// TwinCAT 3 PLC project VekSi_PLC
// ProgramVersion: 3.1.4026.22
// libraries:
//   Tc2_MC2, * (Beckhoff Automation GmbH)
//   Tc2_Standard, * (Beckhoff Automation GmbH)
//   Tc2_System, * (Beckhoff Automation GmbH)
//   Tc2_Utilities, * (Beckhoff Automation GmbH)
//   Tc3_IotBase, * (Beckhoff Automation GmbH)
//   Tc3_JsonXml, * (Beckhoff Automation GmbH)
// project tree:
//   Funtions/ FB_CSVLogger.TcPOU, FB_ValveControl.TcPOU (not stored), FB_MqttManager.TcPOU, MAIN.TcPOU
//   / PlcTask.TcTTO
//   State_Var/ E_CSVLogState.TcDUT, E_MqttManagerState.TcDUT, E_SystemState.TcDUT, E_ValveSource.TcDUT, E_ValveState.TcDUT, ST_MqttConfig.TcDUT, ST_MQTT_Command.TcDUT (not stored), ST_ValveData.TcDUT
//   Variables_Lists/ GVL_Config.TcGVL, GVL_HMI.TcGVL (not stored), GVL_IO.TcGVL, GVL_System.TcGVL (not stored)
// real-time tasks:
//   TASK PlcTask: cycle T#10ms, priority 20, ADS port 350
// motion (NC):
//   TASK NC-Task 1 SAF: cycle T#2ms, priority 4, ADS port 501
//   TASK NC-Task 1 SVB: cycle T#10ms, priority 8, ADS port 511
//   AXIS Axis 2 (id 2)
//     Dynamic: Acceleration=16.9085, Deceleration=16.9085, Jerk=53.5391
//     Velo: RefSearch=3, RefSync=3, SlowManual=3, FastManual=3, Fast=3, Maximum=6
//     OtherSettings: AllowMotionCmdToSlave=true
//     encoder EncType=1
//       EncPara: ScaleFactorNumerator=0.003048
//         Inc: RefSoftSyncMask=#x0000ffff, HomingSensorSource=1
//         TimeComp: TimeCompMode=1, EncDelayCycles=4
//     drive DrvType=24
//       Analog: VeloReferenz=6.096, TorqueSetpointScale=10, ScaleFactorActTorque=0.1
//       TimeComp: TaskDelayCycles=1
//     controller CtrType=1
//       CtrPara: PriorControlFactor=1
//         PosDiffControl: Enable=false
//         Observer: BandWidth=20
//   AXIS Axis 3 (id 3)
//     Dynamic: Acceleration=16.9085, Deceleration=16.9085, Jerk=53.5391
//     Velo: Maximum=6
//     OtherSettings: AllowMotionCmdToSlave=true
//     encoder EncType=1
//       EncPara: ScaleFactorNumerator=0.003048
//         Inc: RefSoftSyncMask=#x0000ffff
//         TimeComp: TimeCompMode=1, EncDelayCycles=4
//     drive DrvType=24
//       Analog: VeloReferenz=6.096, TorqueSetpointScale=10, ScaleFactorActTorque=0.1
//       TimeComp: TaskDelayCycles=1
//     controller CtrType=1
//       CtrPara: PriorControlFactor=1
//         PosDiffControl: Enable=false
//         Observer: BandWidth=20
//   AXIS Axis 1 (id 1)
//     Dynamic: Acceleration=16.9085, Deceleration=16.9085, Jerk=53.5391
//     Velo: RefSearch=3, RefSync=3, SlowManual=3, FastManual=3, Maximum=6
//     OtherSettings: AllowMotionCmdToSlave=true
//     encoder EncType=1
//       EncPara: ScaleFactorNumerator=0.003048
//         Inc: RefSearchInverse=true, RefSoftSyncMask=#x0000ffff
//         TimeComp: TimeCompMode=1, EncDelayCycles=4
//     drive DrvType=24
//       Analog: VeloReferenz=6.096, TorqueSetpointScale=10, ScaleFactorActTorque=0.1
//       TimeComp: TaskDelayCycles=1
//     controller CtrType=1
//       CtrPara: PriorControlFactor=1
//         PosDiffControl: Enable=false
//         Observer: BandWidth=20
// I/O:
//   DEVICE Device 1 (EtherCAT), AmsNetId 192.168.56.1.2.1
//     Term 1 (EK1200) [EK1200-5000 EtherCAT Power supply (2A E-Bus)]
//       Term 2 (EL6070-0033) [EL6070-0033 1Ch. Licence key terminal, individual licences]
//       Term 3 (EL1859) [EL1859 8Ch. Dig. Input 24V, 3ms, 8Ch. Dig. Output 24V, 0.5A]
//       Term 4 (EL3202) [EL3202 2Ch. Ana. Input PT100 (RTD)]
//       Term 5 (EL1004) [EL1004 4Ch. Dig. Input 24V, 3ms]
//       Term 6 (EL3074) [EL3074 4Ch. Ana. Input +/-10V, +/-20mA]
//       Term 7 (EK1322) [EK1322 2-port EtherCAT P junction with feed-in]
//         Box 8 (EPP7041-1002) [EPP7041-1002 1Ch. Stepper motor output stage (50V, 1.5A)]
//       Term 9 (EK1521-0010) [EK1521-0010 1 port EtherCAT junction (FX-SingleMode)]
//         Term 10 (EK1501-0010) [EK1501-0010 EtherCAT Coupler (2A E-Bus, FX-SingleMode, ID switch)]
//           Term 11 (EL3202) [EL3202 2Ch. Ana. Input PT100 (RTD)]
//           Term 12 (EL1859) [EL1859 8Ch. Dig. Input 24V, 3ms, 8Ch. Dig. Output 24V, 0.5A]
//           Term 13 (EL3074) [EL3074 4Ch. Ana. Input +/-10V, +/-20mA]
//           Term 22 (EL9011) [EL9011 End Terminal]
//       Term 14 (EK1521-0010) [EK1521-0010 1 port EtherCAT junction (FX-SingleMode)]
//         Term 15 (EK1501-0010) [EK1501-0010 EtherCAT Coupler (2A E-Bus, FX-SingleMode, ID switch)]
//           Term 16 (EL3202) [EL3202 2Ch. Ana. Input PT100 (RTD)]
//           Term 17 (EL1004) [EL1004 4Ch. Dig. Input 24V, 3ms]
//           Term 18 (EL3074) [EL3074 4Ch. Ana. Input +/-10V, +/-20mA]
//           Term 19 (EK1322) [EK1322 2-port EtherCAT P junction with feed-in]
//             Box 20 (EPP7041-1002) [EPP7041-1002 1Ch. Stepper motor output stage (50V, 1.5A)]
//             Box 21 (EPP7041-1002) [EPP7041-1002 1Ch. Stepper motor output stage (50V, 1.5A)]
// variable links:
//   NC-Task 1 SAF/Axes/Axis 1 <-> Device 1 (EtherCAT)/Term 1 (EK1200)/Term 7 (EK1322)/Box 8 (EPP7041-1002)
//     Drive/Inputs/In/nState1 @bit 3 <-> STM Status/Status/Error
//     Drive/Inputs/In/nState1 @bit 7 <-> STM Status/Status/Motor stall
//     Drive/Inputs/In/nState1 @bit 5 <-> STM Status/Status/Moving negative
//     Drive/Inputs/In/nState1 @bit 4 <-> STM Status/Status/Moving positive
//     Drive/Inputs/In/nState1 @bit 1 <-> STM Status/Status/Ready
//     Drive/Inputs/In/nState1 <-> STM Status/Status/Ready to enable
//     Drive/Inputs/In/nState1 @bit 6 <-> STM Status/Status/Torque reduced
//     Drive/Inputs/In/nState1 @bit 2 <-> STM Status/Status/Warning
//     Drive/Inputs/In/nState2 @bit 4 <-> STM Status/Status/Digital input 2
//     Drive/Inputs/In/nState2 @bit 5 <-> STM Status/Status/Sync error
//     Drive/Inputs/In/nState2 @bit 7 <-> STM Status/Status/TxPDO Toggle
//     Drive/Inputs/In/nState4 @bit 1 <-> WcState/InputToggle
//     Drive/Inputs/In/nState4 <-> WcState/WcState
//     Drive/Outputs/Out/nCtrl1 <-> STM Control/Control/Enable
//     Drive/Outputs/Out/nCtrl1 @bit 2 <-> STM Control/Control/Reduce torque
//     Drive/Outputs/Out/nCtrl1 @bit 1 <-> STM Control/Control/Reset
//     Drive/Outputs/Out/nCtrl2 @bit 3 <-> STM Control/Control/Digital output 1
//     Drive/Outputs/Out/nDataOut2[0] <-> STM Velocity/Velocity
//   NC-Task 1 SAF/Axes/Axis 2 <-> Device 1 (EtherCAT)/Term 1 (EK1200)/Term 14 (EK1521-0010)/Term 15 (EK1501-0010)/Term 19 (EK1322)/Box 20 (EPP7041-1002)
//     Drive/Inputs/In/nState1 @bit 3 <-> STM Status/Status/Error
//     Drive/Inputs/In/nState1 @bit 7 <-> STM Status/Status/Motor stall
//     Drive/Inputs/In/nState1 @bit 5 <-> STM Status/Status/Moving negative
//     Drive/Inputs/In/nState1 @bit 4 <-> STM Status/Status/Moving positive
//     Drive/Inputs/In/nState1 @bit 1 <-> STM Status/Status/Ready
//     Drive/Inputs/In/nState1 <-> STM Status/Status/Ready to enable
//     Drive/Inputs/In/nState1 @bit 6 <-> STM Status/Status/Torque reduced
//     Drive/Inputs/In/nState1 @bit 2 <-> STM Status/Status/Warning
//     Drive/Inputs/In/nState2 @bit 3 <-> STM Status/Status/Digital input 1
//     Drive/Inputs/In/nState2 @bit 4 <-> STM Status/Status/Digital input 2
//     Drive/Inputs/In/nState2 @bit 5 <-> STM Status/Status/Sync error
//     Drive/Inputs/In/nState2 @bit 7 <-> STM Status/Status/TxPDO Toggle
//     Drive/Inputs/In/nState4 @bit 1 <-> WcState/InputToggle
//     Drive/Inputs/In/nState4 <-> WcState/WcState
//     Drive/Outputs/Out/nCtrl1 <-> STM Control/Control/Enable
//     Drive/Outputs/Out/nCtrl1 @bit 2 <-> STM Control/Control/Reduce torque
//     Drive/Outputs/Out/nCtrl1 @bit 1 <-> STM Control/Control/Reset
//     Drive/Outputs/Out/nCtrl2 @bit 3 <-> STM Control/Control/Digital output 1
//     Drive/Outputs/Out/nDataOut2[0] <-> STM Velocity/Velocity
//     Enc/Inputs/In/nDataIn1[0] <-> ENC Status compact/Counter value
//     Enc/Inputs/In/nDataIn2[0] <-> ENC Status compact/Latch value
//     Enc/Inputs/In/nState1 @bit 4 <-> ENC Status compact/Status/Counter overflow
//     Enc/Inputs/In/nState1 @bit 3 <-> ENC Status compact/Status/Counter underflow
//     Enc/Inputs/In/nState1 @bit 7 <-> ENC Status compact/Status/Extrapolation stall
//     Enc/Inputs/In/nState1 <-> ENC Status compact/Status/Latch C valid
//     Enc/Inputs/In/nState1 @bit 1 <-> ENC Status compact/Status/Latch extern valid
//     Enc/Inputs/In/nState1 @bit 2 <-> ENC Status compact/Status/Set counter done
//     Enc/Inputs/In/nState2 @bit 4 <-> ENC Status compact/Status/Status of extern latch
//     Enc/Inputs/In/nState2 <-> ENC Status compact/Status/Status of input A
//     Enc/Inputs/In/nState2 @bit 1 <-> ENC Status compact/Status/Status of input B
//     Enc/Inputs/In/nState2 @bit 2 <-> ENC Status compact/Status/Status of input C
//     Enc/Inputs/In/nState2 @bit 5 <-> ENC Status compact/Status/Sync error
//     Enc/Inputs/In/nState2 @bit 7 <-> ENC Status compact/Status/TxPDO Toggle
//     Enc/Inputs/In/nState4 @bit 1 <-> WcState/InputToggle
//     Enc/Inputs/In/nState4 <-> WcState/WcState
//     Enc/Outputs/Out/nCtrl1 <-> ENC Control compact/Control/Enable latch C
//     Enc/Outputs/Out/nCtrl1 @bit 3 <-> ENC Control compact/Control/Enable latch extern on negative edge
//     Enc/Outputs/Out/nCtrl1 @bit 1 <-> ENC Control compact/Control/Enable latch extern on positive edge
//     Enc/Outputs/Out/nCtrl1 @bit 2 <-> ENC Control compact/Control/Set counter
//     Enc/Outputs/Out/nDataOut1[0] <-> ENC Control compact/Set counter value
//   NC-Task 1 SAF/Axes/Axis 3 <-> Device 1 (EtherCAT)/Term 1 (EK1200)/Term 14 (EK1521-0010)/Term 15 (EK1501-0010)/Term 19 (EK1322)/Box 21 (EPP7041-1002)
//     Drive/Inputs/In/nState1 @bit 3 <-> STM Status/Status/Error
//     Drive/Inputs/In/nState1 @bit 7 <-> STM Status/Status/Motor stall
//     Drive/Inputs/In/nState1 @bit 5 <-> STM Status/Status/Moving negative
//     Drive/Inputs/In/nState1 @bit 4 <-> STM Status/Status/Moving positive
//     Drive/Inputs/In/nState1 @bit 1 <-> STM Status/Status/Ready
//     Drive/Inputs/In/nState1 <-> STM Status/Status/Ready to enable
//     Drive/Inputs/In/nState1 @bit 6 <-> STM Status/Status/Torque reduced
//     Drive/Inputs/In/nState1 @bit 2 <-> STM Status/Status/Warning
//     Drive/Inputs/In/nState2 @bit 3 <-> STM Status/Status/Digital input 1
//     Drive/Inputs/In/nState2 @bit 4 <-> STM Status/Status/Digital input 2
//     Drive/Inputs/In/nState2 @bit 5 <-> STM Status/Status/Sync error
//     Drive/Inputs/In/nState2 @bit 7 <-> STM Status/Status/TxPDO Toggle
//     Drive/Inputs/In/nState4 @bit 1 <-> WcState/InputToggle
//     Drive/Inputs/In/nState4 <-> WcState/WcState
//     Drive/Outputs/Out/nCtrl1 <-> STM Control/Control/Enable
//     Drive/Outputs/Out/nCtrl1 @bit 2 <-> STM Control/Control/Reduce torque
//     Drive/Outputs/Out/nCtrl1 @bit 1 <-> STM Control/Control/Reset
//     Drive/Outputs/Out/nCtrl2 @bit 3 <-> STM Control/Control/Digital output 1
//     Drive/Outputs/Out/nDataOut2[0] <-> STM Velocity/Velocity
//     Enc/Inputs/In/nDataIn1[0] <-> ENC Status compact/Counter value
//     Enc/Inputs/In/nDataIn2[0] <-> ENC Status compact/Latch value
//     Enc/Inputs/In/nState1 @bit 4 <-> ENC Status compact/Status/Counter overflow
//     Enc/Inputs/In/nState1 @bit 3 <-> ENC Status compact/Status/Counter underflow
//     Enc/Inputs/In/nState1 @bit 7 <-> ENC Status compact/Status/Extrapolation stall
//     Enc/Inputs/In/nState1 <-> ENC Status compact/Status/Latch C valid
//     Enc/Inputs/In/nState1 @bit 1 <-> ENC Status compact/Status/Latch extern valid
//     Enc/Inputs/In/nState1 @bit 2 <-> ENC Status compact/Status/Set counter done
//     Enc/Inputs/In/nState2 @bit 4 <-> ENC Status compact/Status/Status of extern latch
//     Enc/Inputs/In/nState2 <-> ENC Status compact/Status/Status of input A
//     Enc/Inputs/In/nState2 @bit 1 <-> ENC Status compact/Status/Status of input B
//     Enc/Inputs/In/nState2 @bit 2 <-> ENC Status compact/Status/Status of input C
//     Enc/Inputs/In/nState2 @bit 5 <-> ENC Status compact/Status/Sync error
//     Enc/Inputs/In/nState2 @bit 7 <-> ENC Status compact/Status/TxPDO Toggle
//     Enc/Inputs/In/nState4 @bit 1 <-> WcState/InputToggle
//     Enc/Inputs/In/nState4 <-> WcState/WcState
//     Enc/Outputs/Out/nCtrl1 <-> ENC Control compact/Control/Enable latch C
//     Enc/Outputs/Out/nCtrl1 @bit 3 <-> ENC Control compact/Control/Enable latch extern on negative edge
//     Enc/Outputs/Out/nCtrl1 @bit 1 <-> ENC Control compact/Control/Enable latch extern on positive edge
//     Enc/Outputs/Out/nCtrl1 @bit 2 <-> ENC Control compact/Control/Set counter
//     Enc/Outputs/Out/nDataOut1[0] <-> ENC Control compact/Set counter value
//   VekSi_PLC/VekSi_PLC Instance <-> Device 1 (EtherCAT)/Term 1 (EK1200)/Term 7 (EK1322)/Box 8 (EPP7041-1002)
//     PlcTask Inputs/GVL_IO.bBottom_position_1 <-> STM Status/Status/Digital input 1
//   VekSi_PLC/VekSi_PLC Instance <-> NC-Task 1 SAF/Axes/Axis 1
//     PlcTask Inputs/MAIN.Axis_Valve1.NcToPlc <-> Outputs/ToPlc
//     PlcTask Outputs/MAIN.Axis_Valve1.PlcToNc <-> Inputs/FromPlc
//   VekSi_PLC/VekSi_PLC Instance <-> NC-Task 1 SAF/Axes/Axis 2
//     PlcTask Inputs/MAIN.Axis_Valve2.NcToPlc <-> Outputs/ToPlc
//     PlcTask Outputs/MAIN.Axis_Valve2.PlcToNc <-> Inputs/FromPlc
//   VekSi_PLC/VekSi_PLC Instance <-> NC-Task 1 SAF/Axes/Axis 3
//     PlcTask Inputs/MAIN.Axis_Valve3.NcToPlc <-> Outputs/ToPlc
//     PlcTask Outputs/MAIN.Axis_Valve3.PlcToNc <-> Inputs/FromPlc

CONFIGURATION VekSi_PLC
    RESOURCE PLC ON TwinCAT3
        TASK PlcTask(INTERVAL := T#10ms, PRIORITY := 20);
        PROGRAM MAIN WITH PlcTask : MAIN;
    END_RESOURCE
END_CONFIGURATION

// ---- State_Var/E_CSVLogState.TcDUT

// States:
//   CSV_IDLE        : Waiting for next log interval
//   CSV_PREPARE     : Build timestamp, filename, header/row strings
//   CSV_OPEN        : Open file in append mode
//   CSV_WRITE_HDR   : Write header (first row for new day in this PLC session)
//   CSV_WRITE_ROW   : Write one CSV data row
//   CSV_CLOSE       : Close file handle
//   CSV_ERROR       : Latch error until disabled or reset by logic
// ============================================================
TYPE E_CSVLogState :
(
    CSV_IDLE      := 0,
    CSV_PREPARE   := 1,
    CSV_OPEN      := 2,
    CSV_WRITE_HDR := 3,
    CSV_WRITE_ROW := 4,
    CSV_CLOSE     := 5,
    CSV_ERROR     := 6
);
END_TYPE

// ---- State_Var/E_MqttManagerState.TcDUT
{attribute 'strict'}
{attribute 'to_string'}
TYPE E_MqttManagerState :
(
    DISABLED        := 0,
    CONNECTING      := 1,
    CONNECTED       := 2,
    DISCONNECTING   := 3,
    WAIT_RECONNECT  := 4
);
END_TYPE

// ---- State_Var/E_SystemState.TcDUT
{attribute 'strict'}
{attribute 'to_string'}
TYPE E_SystemState :
(
    INIT             := 0,
    HOMING_REQUIRED  := 1,
    READY            := 2,
    RUN              := 3,
    FAULT            := 4
);
END_TYPE

// ---- State_Var/E_ValveSource.TcDUT
{attribute 'qualified_only'}
{attribute 'strict'}
{attribute 'to_string'}
TYPE E_ValveSource :
(
    NONE    := 0,   // No command received yet (startup default)
    HMI     := 1,   // Last setpoint was entered via local HMI
    MQTT    := 2    // Last setpoint was received via MQTT topic
);
END_TYPE

// ---- State_Var/E_ValveState.TcDUT
{attribute 'qualified_only'}
{attribute 'strict'}
{attribute 'to_string'}
TYPE E_ValveState :
(
    INIT    := 0,   // Initializing, powering axis
    HOMING  := 1,   // Performing homing sequence (MC_Home)
    IDLE    := 2,   // At position, no active command
    MOVING  := 3,   // MC_MoveAbsolute active, travelling to setpoint
	HALT	:= 4,
    HOLD    := 5,   // At setpoint, holding position
    FAULT   := 6,   // Error state — MC error, drive fault, or limit breach
    RESET   := 7    // Clearing fault, preparing to re-home
);
END_TYPE

// ---- State_Var/ST_MqttConfig.TcDUT
(*
  ST_MqttConfig
  =============
  Central MQTT runtime configuration structure.

  Project policy (this project):
  - Broker and topic settings are maintained in PLC code constants (GVL_Config).
  - HMI only enables/disables MQTT operation.
  - No broker parameter editing from HMI.
*)
TYPE ST_MqttConfig :
STRUCT
  (* ── Broker connection parameters ────────────────────────── *)
  sBrokerAddress  : STRING(255);   (* IP/hostname of broker                        *)
  nPort           : UINT;          (* 1883 = plain MQTT, 8883 = TLS (if enabled)   *)
  sClientId       : STRING(64);    (* Must be unique per broker                    *)
  sUsername       : STRING(64);    (* Optional                                      *)
  sPassword       : STRING(64);    (* Optional                                      *)
  bUseTls         : BOOL;          (* TRUE = secure transport (if broker supports)  *)

  (* ── Topic parameters ────────────────────────────────────── *)
  sTopicPrefix    : STRING(64);    (* Logical namespace, e.g. 'irrigation/site1'   *)
  sMainTopic      : STRING(128);   (* Status publish topic                          *)
  SubscribeTopic  : STRING(128);   (* Command subscribe topic                       *)

  (* ── Runtime timings ─────────────────────────────────────── *)
  tPublishInterval : TIME;         (* Periodic status publish interval              *)
  tReconnectDelay  : TIME;         (* Delay between reconnect attempts              *)
END_STRUCT
END_TYPE

// ---- State_Var/ST_ValveData.TcDUT

TYPE ST_ValveData :
STRUCT
    // --- Setpoints (written by HMI or MQTT) ---
    HMI_Setpoint    : REAL;         // Position setpoint from HMI (0.0–100.0 %)
    MQTT_Setpoint   : REAL;         // Position setpoint from MQTT (0.0–100.0 %)
    Active_Setpoint : REAL;         // Currently active setpoint (latest of HMI/MQTT)

    // --- Feedback (written by FB_ValveControl) ---
    Actual_Position : REAL;         // Actual valve position in % (from MC axis)
    Actual_Pos_Raw  : LREAL;        // Raw axis position in mm or steps (from MC2)

    // --- Command source tracking ---
    Source          : E_ValveSource;  // Who issued the last command
    MQTT_Enabled    : BOOL;           // Allow MQTT to override this valve's setpoint

    // --- State machine status ---
    State           : E_ValveState;  // Current state of FB_ValveControl
    IsHomed         : BOOL;          // TRUE once homing has been completed
    InPosition      : BOOL;          // TRUE when actual ≈ setpoint (within tolerance)
    IsFault         : BOOL;          // TRUE when in FAULT state
    FaultCode       : UDINT;         // MC or drive error code for diagnostics
	

	
    // --- Reset ---
    Reset_Cmd       : BOOL;          // HMI writes TRUE to request fault reset
END_STRUCT
END_TYPE

// ---- Variables_Lists/GVL_Config.TcGVL
{attribute 'qualified_only'}
VAR_GLOBAL CONSTANT
    // ── Valve motion parameters ───────────────────────────────
    VALVE_FULL_STROKE_MM           : REAL  := 6.096;     // Mechanical full travel for 0..100% scaling
    VALVE_POSITION_TOLERANCE       : REAL  := 0.5;       // In-position dead-band in percent
    VALVE_MOVE_VELOCITY            : LREAL := 1.5;       // mm/s
    VALVE_MOVE_ACCELERATION        : LREAL := 16.9085;   // mm/s²
    VALVE_MOVE_DECELERATION        : LREAL := 16.9085;   // mm/s²
    VALVE_MOVE_JERK                : LREAL := 53.5391;   // mm/s³
    VALVE_HOMING_VELOCITY          : LREAL := 1.0;       // Reference only (NC axis settings still apply)

    // ── CSV Logging ───────────────────────────────────────────
    CSV_LOG_INTERVAL_S             : TIME   := T#15M;
    CSV_FILE_PATH                  : STRING := 'C:\TwinCAT\3.1\Boot\Log\';
    CSV_FILENAME_PREFIX            : STRING := 'IrrigationLog_';

    // ── MQTT defaults (single source of truth) ───────────────
    // All MQTT configuration is centralized in this one constant structure.
    MQTT_CONFIG : ST_MqttConfig := (
        sBrokerAddress   := '192.168.1.100',
        nPort            := 1883,
        sClientId        := 'BeckhoffIrrigationPLC',
        sUsername        := '',
        sPassword        := '',
        bUseTls          := FALSE,
        sTopicPrefix     := 'irrigation',
        sMainTopic       := 'irrigation/status',
        SubscribeTopic   := 'irrigation/command',
        tPublishInterval := T#5M,
        tReconnectDelay  := T#30S
    );

    // ── Task cycle time ───────────────────────────────────────
    TASK_CYCLE_MS                  : UINT := 10;         // Must match TwinCAT task setting
END_VAR

// ---- Variables_Lists/GVL_IO.TcGVL
{attribute 'qualified_only'}
VAR_GLOBAL
	
	AI_L1V11  			: INT	:= -999 ;	// AT %I* // Water Level Sensors
	AI_L1V20  			: INT	:= -999 ;	// AT %I*
	AI_L2V21  			: INT	:= -999 ;	// AT %I*

	AI_Tmp_1 			: INT	:= -999;	// AT %I*
	AI_Tmp_2  			: INT	:= -999;	// AT %I*
	
	AI_PosFeedback_1	: INT	:= -999;	// AT %I* //Position feedback from the encoder
	AI_PosFeedback_2	: INT	:= -999;	// AT %I*
	AI_PosFeedback_3	: INT	:= -999;	// AT %I*
	

	bTop_position_1		AT %I*	: BOOL;
	bBottom_position_1	AT %I*	: BOOL;
END_VAR

// ---- Funtions/MAIN.TcPOU
PROGRAM MAIN
VAR
    // ── Valve function blocks (one instance per physical axis) ───────────────────
    fbValve1    : FB_ValveControl;
    fbValve2    : FB_ValveControl;
    fbValve3    : FB_ValveControl;

    // ── NC axis references ─────────────────────────────────────────────────────────
    // These variables must be linked to configured TwinCAT NC axes in I/O mapping.
    Axis_Valve1 : AXIS_REF;
    Axis_Valve2 : AXIS_REF;
    Axis_Valve3 : AXIS_REF;

    // ── Supporting modules ─────────────────────────────────────────────────────────
    fbCsvLogger   : FB_CsvLogger;
    fbMqttManager : FB_MqttManager;

    // ── MQTT runtime configuration ─────────────────────────────────────────────────
    // Initialized from GVL_Config once at startup. Fields may be changed in code
    // later if dynamic reconfiguration from HMI is added.
    stMqttConfig : ST_MqttConfig := (
        sBrokerAddress := GVL_Config.MQTT_DEFAULT_BROKER_IP,
        nPort := GVL_Config.MQTT_DEFAULT_PORT,
        sClientId := GVL_Config.MQTT_DEFAULT_CLIENT_ID,
        sUsername := GVL_Config.MQTT_DEFAULT_USERNAME,
        sPassword := GVL_Config.MQTT_DEFAULT_PASSWORD,
        sTopicPrefix := GVL_Config.MQTT_DEFAULT_TOPIC_PREFIX,
        sMainTopic := 'irrigation/status',
        SubscribeTopic := 'irrigation/command',
        tPublishInterval := T#5M,
        tReconnectDelay := T#30S
    );

    // ── Command arbitration helpers ────────────────────────────────────────────────
    // Stores previous HMI setpoints to detect operator changes.
    arrPrevHmiSetpoint : ARRAY[1..3] OF REAL := [-1.0, -1.0, -1.0];

    // Arrays passed directly to MQTT manager for compact status publishing.
    arrValveSetpoint : ARRAY[1..3] OF REAL;
    arrValveActual   : ARRAY[1..3] OF REAL;
    arrValveSource   : ARRAY[1..3] OF STRING(32);

    // Generic loop index used for repetitive valve operations.
    iValve : INT;
END_VAR

// =============================================================================
// SECTION 1 — READ HMI INPUTS AND CLAMP OPERATOR SETPOINTS
// =============================================================================
// LIMIT guarantees every valve command remains inside the configured legal range.
GVL_System.Valve[1].HMI_Setpoint := LIMIT(0.0, GVL_HMI.HMI_Valve1_Setpoint, 100.0);
GVL_System.Valve[2].HMI_Setpoint := LIMIT(0.0, GVL_HMI.HMI_Valve2_Setpoint, 100.0);
GVL_System.Valve[3].HMI_Setpoint := LIMIT(0.0, GVL_HMI.HMI_Valve3_Setpoint, 100.0);

GVL_System.Valve[1].Reset_Cmd := GVL_HMI.HMI_Valve1_Reset;
GVL_System.Valve[2].Reset_Cmd := GVL_HMI.HMI_Valve2_Reset;
GVL_System.Valve[3].Reset_Cmd := GVL_HMI.HMI_Valve3_Reset;

IF GVL_HMI.HMI_ResetAll THEN
    // Global reset request from HMI: pulse every valve reset command in this cycle.
    FOR iValve := 1 TO 3 DO
        GVL_System.Valve[iValve].Reset_Cmd := TRUE;
    END_FOR
    GVL_HMI.HMI_ResetAll := FALSE;
END_IF


// =============================================================================
// SECTION 2 — SETPOINT SOURCE ARBITRATION (HMI vs MQTT)
// =============================================================================
FOR iValve := 1 TO 3 DO
    // Startup fallback: if source is unknown, default to local HMI control.
    IF GVL_System.Valve[iValve].Source = E_ValveSource.NONE THEN
        GVL_System.Valve[iValve].Source := E_ValveSource.HMI;
        GVL_System.Valve[iValve].Active_Setpoint := GVL_System.Valve[iValve].HMI_Setpoint;
    END_IF

    // When operator changes HMI setpoint, HMI becomes authoritative source.
    IF ABS(GVL_System.Valve[iValve].HMI_Setpoint - arrPrevHmiSetpoint[iValve]) > 0.001 THEN
        GVL_System.Valve[iValve].Active_Setpoint := GVL_System.Valve[iValve].HMI_Setpoint;
        GVL_System.Valve[iValve].Source := E_ValveSource.HMI;
        arrPrevHmiSetpoint[iValve] := GVL_System.Valve[iValve].HMI_Setpoint;
    END_IF

    // Build compact telemetry arrays once here (reused by MQTT manager call).
    arrValveSetpoint[iValve] := GVL_System.Valve[iValve].Active_Setpoint;
    arrValveActual[iValve] := GVL_System.Valve[iValve].Actual_Position;
    arrValveSource[iValve] := TO_STRING(GVL_System.Valve[iValve].Source);
END_FOR


// =============================================================================
// SECTION 3 — MQTT CLIENT HANDLING
// =============================================================================
fbMqttManager (
    bEnable               := GVL_HMI.HMI_MQTT_bEnable,
    stConfig              := stMqttConfig,
    bApplyConfig          := FALSE,
    bPublish              := GVL_HMI.HMI_MQTT_mPublish,
    sPubTopic             := stMqttConfig.sMainTopic,
    sPubPayload           := '',
    bSubscribe            := GVL_HMI.HMI_MQTT_bEnable,
    sSubTopic             := stMqttConfig.SubscribeTopic,
    bUnsubscribe          := FALSE,
    sUnsubTopic           := '',
    bEnableStatusPublish  := GVL_HMI.HMI_MQTT_bEnable,
    tStatusPublishTime    := T#5M,
    sStatusTopic          := stMqttConfig.sMainTopic,
    rValveSetpoint        := arrValveSetpoint,
    rValveActual          := arrValveActual,
    sValveSource          := arrValveSource,
    rTemperature_C        := INT_TO_REAL(GVL_IO.AI_Tmp_1),
    rWaterLevel_Percent   := INT_TO_REAL(GVL_IO.AI_L1V11),
    sTimestamp            := DT_TO_STRING(CURRENT_DT())
);

IF fbMqttManager.bNewRemoteCommand AND GVL_HMI.HMI_MQTT_bEnable THEN
    // Remote command became valid in this cycle. Clamp values for safety before use.
    FOR iValve := 1 TO 3 DO
        GVL_System.Valve[iValve].MQTT_Setpoint := LIMIT(0.0, fbMqttManager.rMqttValveSetpoint[iValve], 100.0);
        GVL_System.Valve[iValve].Active_Setpoint := GVL_System.Valve[iValve].MQTT_Setpoint;
        GVL_System.Valve[iValve].Source := E_ValveSource.MQTT;
    END_FOR
END_IF


// =============================================================================
// SECTION 4 — EXECUTE PER-VALVE CONTROL FBs
// =============================================================================
// NOTE: Each valve FB is explicit to keep wiring to dedicated HMI tags readable.

// ── Valve 1 ────────────────────────────────────────────────────────────────────
fbValve1(
    Axis            := Axis_Valve1,
    HMI_Setpoint    := GVL_System.Valve[1].HMI_Setpoint,
    MQTT_Setpoint   := GVL_System.Valve[1].MQTT_Setpoint,
    MQTT_Enabled    := GVL_HMI.HMI_MQTT_bEnable,
    Enable          := TRUE,
    eHomingSelection := MC_Direct,
    Reset           := GVL_System.Valve[1].Reset_Cmd,
    MoveVelocity    := GVL_Config.VALVE_MOVE_VELOCITY,
    MoveAccel       := GVL_Config.VALVE_MOVE_ACCELERATION,
    MoveDecel       := GVL_Config.VALVE_MOVE_DECELERATION,
    MoveJerk        := GVL_Config.VALVE_MOVE_JERK,
    HomeVelocity    := GVL_Config.VALVE_HOMING_VELOCITY,
    FullStroke_mm   := GVL_Config.VALVE_FULL_STROKE_MM,
    PosTolerance    := GVL_Config.VALVE_POSITION_TOLERANCE,
    Move_Stop       := GVL_HMI.HMI_Valve1_Stop,
    UPDATE          := GVL_HMI.HMI_UPDATE,
    ZeroPosition    := GVL_IO.bBottom_position_1,
    bHoming         := GVL_HMI.HMI_Valve1_Homing,

    Actual_Position => GVL_System.Valve[1].Actual_Position,
    State           => GVL_System.Valve[1].State,
    Source          => GVL_System.Valve[1].Source,
    IsHomed         => GVL_System.Valve[1].IsHomed,
    InPosition      => GVL_System.Valve[1].InPosition,
    IsFault         => GVL_System.Valve[1].IsFault,
    FaultCode       => GVL_System.Valve[1].FaultCode,

    rTarget_mm      => GVL_HMI.Raw_Valve1_Setpoint,
    rActual_mm      => GVL_HMI.Raw_Valve1_Position
);

// ── Valve 2 ────────────────────────────────────────────────────────────────────
fbValve2(
    Axis            := Axis_Valve2,
    HMI_Setpoint    := GVL_System.Valve[2].HMI_Setpoint,
    MQTT_Setpoint   := GVL_System.Valve[2].MQTT_Setpoint,
    MQTT_Enabled    := GVL_HMI.HMI_MQTT_bEnable,
    Enable          := TRUE,
    eHomingSelection := MC_Direct,
    Reset           := GVL_System.Valve[2].Reset_Cmd,
    MoveVelocity    := GVL_Config.VALVE_MOVE_VELOCITY,
    MoveAccel       := GVL_Config.VALVE_MOVE_ACCELERATION,
    MoveDecel       := GVL_Config.VALVE_MOVE_DECELERATION,
    MoveJerk        := GVL_Config.VALVE_MOVE_JERK,
    HomeVelocity    := GVL_Config.VALVE_HOMING_VELOCITY,
    FullStroke_mm   := GVL_Config.VALVE_FULL_STROKE_MM,
    PosTolerance    := GVL_Config.VALVE_POSITION_TOLERANCE,
    Move_Stop       := GVL_HMI.HMI_Valve2_Stop,
    UPDATE          := GVL_HMI.HMI_UPDATE,
    bHoming         := GVL_HMI.HMI_Valve2_Homing,

    Actual_Position => GVL_System.Valve[2].Actual_Position,
    State           => GVL_System.Valve[2].State,
    Source          => GVL_System.Valve[2].Source,
    IsHomed         => GVL_System.Valve[2].IsHomed,
    InPosition      => GVL_System.Valve[2].InPosition,
    IsFault         => GVL_System.Valve[2].IsFault,
    FaultCode       => GVL_System.Valve[2].FaultCode,

    rTarget_mm      => GVL_HMI.Raw_Valve2_Setpoint,
    rActual_mm      => GVL_HMI.Raw_Valve2_Position
);

// ── Valve 3 ────────────────────────────────────────────────────────────────────
fbValve3(
    Axis            := Axis_Valve3,
    HMI_Setpoint    := GVL_System.Valve[3].HMI_Setpoint,
    MQTT_Setpoint   := GVL_System.Valve[3].MQTT_Setpoint,
    MQTT_Enabled    := GVL_HMI.HMI_MQTT_bEnable,
    Enable          := TRUE,
    eHomingSelection := MC_Direct,
    Reset           := GVL_System.Valve[3].Reset_Cmd,
    MoveVelocity    := GVL_Config.VALVE_MOVE_VELOCITY,
    MoveAccel       := GVL_Config.VALVE_MOVE_ACCELERATION,
    MoveDecel       := GVL_Config.VALVE_MOVE_DECELERATION,
    MoveJerk        := GVL_Config.VALVE_MOVE_JERK,
    HomeVelocity    := GVL_Config.VALVE_HOMING_VELOCITY,
    FullStroke_mm   := GVL_Config.VALVE_FULL_STROKE_MM,
    PosTolerance    := GVL_Config.VALVE_POSITION_TOLERANCE,
    Move_Stop       := GVL_HMI.HMI_Valve3_Stop,
    UPDATE          := GVL_HMI.HMI_UPDATE,
    bHoming         := GVL_HMI.HMI_Valve3_Homing,

    Actual_Position => GVL_System.Valve[3].Actual_Position,
    State           => GVL_System.Valve[3].State,
    Source          => GVL_System.Valve[3].Source,
    IsHomed         => GVL_System.Valve[3].IsHomed,
    InPosition      => GVL_System.Valve[3].InPosition,
    IsFault         => GVL_System.Valve[3].IsFault,
    FaultCode       => GVL_System.Valve[3].FaultCode,

    rTarget_mm      => GVL_HMI.Raw_Valve3_Setpoint,
    rActual_mm      => GVL_HMI.Raw_Valve3_Position
);


// =============================================================================
// SECTION 5 — CSV LOGGER EXECUTION
// =============================================================================
fbCsvLogger(
    bEnable              := TRUE,
    bForceWrite          := GVL_HMI.WriteTrigger,
    tLogInterval         := GVL_Config.CSV_LOG_INTERVAL_S,
    sBasePath            := GVL_Config.CSV_FILE_PATH,
    sPrefix              := GVL_Config.CSV_FILENAME_PREFIX,
    stValve              := GVL_System.Valve,
    rWaterLevel_Percent  := INT_TO_REAL(GVL_IO.AI_L1V11),
    rTemperature_C       := INT_TO_REAL(GVL_IO.AI_Tmp_1),

    dtLastWrite          => GVL_System.CSV_LastWriteTime,
    bError               => GVL_System.CSV_FileError,
    sCurrentFilename     => GVL_System.CSV_CurrentFile,
    eState               => GVL_System.CSV_LoggerState
);


// =============================================================================
// SECTION 6 — CLEANUP + HMI MIRRORING
// =============================================================================
// Reset commands are pulse-based: clear them after handing to FBs.
FOR iValve := 1 TO 3 DO
    GVL_System.Valve[iValve].Reset_Cmd := FALSE;
END_FOR
GVL_HMI.HMI_Valve1_Reset := FALSE;
GVL_HMI.HMI_Valve2_Reset := FALSE;
GVL_HMI.HMI_Valve3_Reset := FALSE;

// Copy valve runtime status to HMI tags.
GVL_HMI.ACT_Valve1_Position  := GVL_System.Valve[1].Actual_Position;
GVL_HMI.ACT_Valve1_State     := GVL_System.Valve[1].State;
GVL_HMI.ACT_Valve1_Source    := GVL_System.Valve[1].Source;
GVL_HMI.ACT_Valve1_Fault     := GVL_System.Valve[1].IsFault;
GVL_HMI.ACT_Valve1_FaultCode := GVL_System.Valve[1].FaultCode;

GVL_HMI.ACT_Valve2_Position  := GVL_System.Valve[2].Actual_Position;
GVL_HMI.ACT_Valve2_State     := GVL_System.Valve[2].State;
GVL_HMI.ACT_Valve2_Source    := GVL_System.Valve[2].Source;
GVL_HMI.ACT_Valve2_Fault     := GVL_System.Valve[2].IsFault;
GVL_HMI.ACT_Valve2_FaultCode := GVL_System.Valve[2].FaultCode;

GVL_HMI.ACT_Valve3_Position  := GVL_System.Valve[3].Actual_Position;
GVL_HMI.ACT_Valve3_State     := GVL_System.Valve[3].State;
GVL_HMI.ACT_Valve3_Source    := GVL_System.Valve[3].Source;
GVL_HMI.ACT_Valve3_Fault     := GVL_System.Valve[3].IsFault;
GVL_HMI.ACT_Valve3_FaultCode := GVL_System.Valve[3].FaultCode;

// System readiness is true only when all valves are homed and fault free.
GVL_System.AnyFaultActive :=
    GVL_System.Valve[1].IsFault OR
    GVL_System.Valve[2].IsFault OR
    GVL_System.Valve[3].IsFault;

GVL_System.SystemReady :=
    GVL_System.Valve[1].IsHomed AND
    GVL_System.Valve[2].IsHomed AND
    GVL_System.Valve[3].IsHomed AND
    NOT GVL_System.AnyFaultActive;

GVL_HMI.ACT_SystemReady := GVL_System.SystemReady;

END_PROGRAM

// ---- Funtions/FB_CSVLogger.TcPOU
(*  FB_CsvLogger
  ============
  Writes valve and sensor snapshots to CSV files on the IPC filesystem.

  File naming:
    <BasePath><Prefix><YYYY-MM-DD>.csv
  Example:
    C:\TwinCAT\IrrigationLogs\Irrigation_2026-04-28.csv

  Why a state machine?
    TwinCAT file function blocks are asynchronous (non-blocking). Each file
    action may require several PLC cycles to complete. This FB advances through
    explicit states so it remains deterministic and easy to troubleshoot.
*)

FUNCTION_BLOCK FB_CsvLogger

VAR_INPUT
  bEnable              : BOOL := TRUE;
  bForceWrite          : BOOL;          (* Rising edge = write one row immediately    *)
  tLogInterval         : TIME;          (* Periodic write interval                     *)
  sBasePath            : STRING(128);   (* Folder path including trailing '\'         *)
  sPrefix              : T_MaxString;   (* File prefix, e.g. 'Irrigation_'             *)
  stValve              : ARRAY[1..3] OF ST_ValveData;
  rWaterLevel_Percent  : REAL;
  rTemperature_C       : REAL;
END_VAR

VAR_OUTPUT
  bBusy                : BOOL;
  bError               : BOOL;
  nErrorCode           : UDINT;
  bFileExists          : BOOL := FALSE;
  dtLastWrite          : DT;
  sCurrentFile         : STRING(128);
  sCurrentFilename     : STRING(128);
  eState               : E_CSVLogState := E_CSVLogState.CSV_IDLE;
END_VAR

VAR
  (* ── File I/O FBs ───────────────────────────────────────── *)
  fbFileOpen           : FB_FileOpen;
  fbFileWrite          : FB_FileWrite;
  fbFileClose          : FB_FileClose;
  fbEnum               : FB_EnumFindFileEntry;

  hFilenumber          : UINT;
  cbLen                : UDINT;

  (* ── Trigger handling ───────────────────────────────────── *)
  tIntervalTimer       : TON;
  rtForceWrite         : R_TRIG;
  bTriggerWrite        : BOOL;

  (* ── Time/date helpers ──────────────────────────────────── *)
  fbGetTime            : FB_LocalSystemTime;
  nYear                : UINT;
  nMonth               : UINT;
  nDay                 : UINT;
  sYear                : STRING(8);
  sMonth               : STRING(4);
  sDay                 : STRING(4);

  (* ── CSV string buffers ─────────────────────────────────── *)
  sLine                : STRING(512);
  sHeader              : STRING(512);
  sSource              : STRING(8);

  (* ── Internal state helpers ─────────────────────────────── *)
  bEnumStart           : BOOL;
END_VAR

(* ============================================================
   SECTION 1 — CYCLIC HOUSEKEEPING
   ============================================================ *)
fbGetTime(bEnable := TRUE, dwCycle := 1);

// If logger is disabled, remain safe and idle.
IF NOT bEnable THEN
  tIntervalTimer(IN := FALSE);
  bTriggerWrite := FALSE;
  bBusy := FALSE;

  IF hFilenumber <> 0 THEN
    // Close any leftover open file handle before returning to idle.
    fbFileClose(hFile := hFilenumber, bExecute := TRUE);
    IF NOT fbFileClose.bBusy THEN
      fbFileClose(bExecute := FALSE);
      hFilenumber := 0;
    END_IF
  END_IF

  eState := E_CSVLogState.CSV_IDLE;
  RETURN;
END_IF

rtForceWrite(CLK := bForceWrite);
tIntervalTimer(IN := TRUE, PT := tLogInterval);

bTriggerWrite := rtForceWrite.Q OR tIntervalTimer.Q;

IF tIntervalTimer.Q THEN
  // Retrigger periodic timer after each elapsed interval.
  tIntervalTimer(IN := FALSE);
END_IF


(* ============================================================
   SECTION 2 — LOGGER STATE MACHINE
   ============================================================ *)
CASE eState OF

  E_CSVLogState.CSV_IDLE:
    bBusy := FALSE;

    IF bTriggerWrite THEN
      bError := FALSE;
      nErrorCode := 0;
      bFileExists := FALSE;
      bEnumStart := TRUE;
      eState := E_CSVLogState.CSV_PREPARE;
    END_IF


  E_CSVLogState.CSV_PREPARE:
    // Build filename as Prefix + YYYY-MM-DD.csv (daily file rotation).
    nYear  := fbGetTime.systemTime.wYear;
    nMonth := fbGetTime.systemTime.wMonth;
    nDay   := fbGetTime.systemTime.wDay;

    sYear  := UINT_TO_STRING(nYear);
    sMonth := UINT_TO_STRING(nMonth);
    sDay   := UINT_TO_STRING(nDay);

    IF nMonth < 10 THEN
      sMonth := CONCAT('0', sMonth);
    END_IF

    IF nDay < 10 THEN
      sDay := CONCAT('0', sDay);
    END_IF

    sCurrentFilename := sPrefix;
    sCurrentFilename := CONCAT(sCurrentFilename, sYear);
    sCurrentFilename := CONCAT(sCurrentFilename, '-');
    sCurrentFilename := CONCAT(sCurrentFilename, sMonth);
    sCurrentFilename := CONCAT(sCurrentFilename, '-');
    sCurrentFilename := CONCAT(sCurrentFilename, sDay);
    sCurrentFilename := CONCAT(sCurrentFilename, '.csv');

    sCurrentFile := CONCAT(sBasePath, sCurrentFilename);

    // Determine whether file already exists (header needed only for new files).
    IF bEnumStart THEN
      fbEnum(
        sPathName := sCurrentFile,
        eCmd := eEnumCmd_First,
        bExecute := TRUE,
        tTimeout := T#2S
      );
      bEnumStart := FALSE;
    ELSE
      fbEnum(bExecute := FALSE);
    END_IF

    IF NOT fbEnum.bBusy THEN
      fbEnum(bExecute := FALSE);

      IF (NOT fbEnum.bError) AND (fbEnum.stFindFile.sFileName <> '') THEN
        bFileExists := TRUE;
      ELSE
        bFileExists := FALSE;
      END_IF

      eState := E_CSVLogState.CSV_OPEN;
    END_IF


  E_CSVLogState.CSV_OPEN:
    bBusy := TRUE;

    fbFileOpen(
      sPathName := sCurrentFile,
      nMode     := FOPEN_MODEAPPEND,
      bExecute  := TRUE,
      hFile     => hFilenumber
    );

    IF NOT fbFileOpen.bBusy THEN
      fbFileOpen(bExecute := FALSE);

      IF fbFileOpen.bError THEN
        nErrorCode := fbFileOpen.nErrId;
        bError := TRUE;
        eState := E_CSVLogState.CSV_ERROR;
      ELSE
        hFilenumber := fbFileOpen.hFile;

        IF bFileExists THEN
          eState := E_CSVLogState.CSV_WRITE_ROW;
        ELSE
          eState := E_CSVLogState.CSV_WRITE_HDR;
        END_IF
      END_IF
    END_IF


  E_CSVLogState.CSV_WRITE_HDR:
    // Header is written exactly once per newly created daily file.
    sHeader := 'Timestamp,V1_Setpoint_%,V1_Actual_%,V1_Source,V2_Setpoint_%,V2_Actual_%,V2_Source,V3_Setpoint_%,V3_Actual_%,V3_Source,WaterLevel_%,Temperature_C$R$N';
    cbLen := INT_TO_UDINT(LEN(sHeader));

    fbFileWrite(
      bExecute   := TRUE,
      hFile      := hFilenumber,
      pWriteBuff := ADR(sHeader),
      cbWriteLen := cbLen
    );

    IF NOT fbFileWrite.bBusy THEN
      fbFileWrite(bExecute := FALSE);

      IF fbFileWrite.bError THEN
        nErrorCode := fbFileWrite.nErrId;
        bError := TRUE;
        eState := E_CSVLogState.CSV_CLOSE;
      ELSE
        eState := E_CSVLogState.CSV_WRITE_ROW;
      END_IF
    END_IF


  E_CSVLogState.CSV_WRITE_ROW:
    // Compose one CSV line from the latest process snapshot.
    sLine := CONCAT(SYSTEMTIME_TO_STRING(fbGetTime.systemTime), ',');

    sLine := CONCAT(sLine, CONCAT(REAL_TO_STRING(stValve[1].Active_Setpoint), ','));
    sLine := CONCAT(sLine, CONCAT(REAL_TO_STRING(stValve[1].Actual_Position), ','));
    sSource := TO_STRING(stValve[1].Source);
    sLine := CONCAT(sLine, CONCAT(sSource, ','));

    sLine := CONCAT(sLine, CONCAT(REAL_TO_STRING(stValve[2].Active_Setpoint), ','));
    sLine := CONCAT(sLine, CONCAT(REAL_TO_STRING(stValve[2].Actual_Position), ','));
    sSource := TO_STRING(stValve[2].Source);
    sLine := CONCAT(sLine, CONCAT(sSource, ','));

    sLine := CONCAT(sLine, CONCAT(REAL_TO_STRING(stValve[3].Active_Setpoint), ','));
    sLine := CONCAT(sLine, CONCAT(REAL_TO_STRING(stValve[3].Actual_Position), ','));
    sSource := TO_STRING(stValve[3].Source);
    sLine := CONCAT(sLine, CONCAT(sSource, ','));

    sLine := CONCAT(sLine, CONCAT(REAL_TO_STRING(rWaterLevel_Percent), ','));
    sLine := CONCAT(sLine, CONCAT(REAL_TO_STRING(rTemperature_C), '$R$N'));

    cbLen := INT_TO_UDINT(LEN(sLine));

    fbFileWrite(
      bExecute   := TRUE,
      hFile      := hFilenumber,
      pWriteBuff := ADR(sLine),
      cbWriteLen := cbLen
    );

    IF NOT fbFileWrite.bBusy THEN
      fbFileWrite(bExecute := FALSE);

      IF fbFileWrite.bError THEN
        nErrorCode := fbFileWrite.nErrId;
        bError := TRUE;
      ELSE
        bError := FALSE;
        dtLastWrite := SYSTEMTIME_TO_DT(fbGetTime.systemTime);
      END_IF

      eState := E_CSVLogState.CSV_CLOSE;
    END_IF


  E_CSVLogState.CSV_CLOSE:
    fbFileClose(hFile := hFilenumber, bExecute := TRUE);

    IF NOT fbFileClose.bBusy THEN
      fbFileClose(bExecute := FALSE);
      hFilenumber := 0;
      bBusy := FALSE;
      eState := E_CSVLogState.CSV_IDLE;
    END_IF


  E_CSVLogState.CSV_ERROR:
    bBusy := FALSE;
    bError := TRUE;

    // Recovery strategy: on next trigger, retry from preparation phase.
    IF bTriggerWrite THEN
      eState := E_CSVLogState.CSV_PREPARE;
    END_IF

END_CASE

END_FUNCTION_BLOCK

// ---- Funtions/FB_MqttManager.TcPOU
(*
============================================================
FUNCTION_BLOCK: FB_MqttManager
============================================================

PURPOSE
  Central MQTT manager for irrigation system.

  NOVICE SUMMARY
  - Think of this FB as a communication gateway between PLC and broker.
  - It handles connect/reconnect and topic subscription lifecycle.
  - It converts incoming JSON command payload into valve setpoints.
  - It builds outgoing JSON status payload from PLC runtime values.

HANDLES
  • MQTT connection / reconnection
  • Topic subscription / unsubscription
  • Manual publish
  • Cyclic JSON status publish
  • Incoming JSON command parsing
  • List of currently subscribed topics for HMI

EXPECTED INCOMING JSON
  {
    "valve_1": 25.0,
    "valve_2": 50.0,
    "valve_3": 75.0
  }

OUTGOING JSON
  Similar to CSV row:
    timestamp,
    valve setpoints,
    valve actual positions,
    valve command sources,
    temperature,
    water level

LIBRARIES
  • TF6701 / Tc3_IotBase
  • Tc2_Standard
============================================================
*)

FUNCTION_BLOCK FB_MqttManager
VAR_INPUT
    (* ── Connection control ───────────────────────────── *)
    bEnable         : BOOL;             (* Master enable. FALSE disconnects MQTT. *)
    stConfig        : ST_MqttConfig;    (* Broker address, port, username, etc.   *)
    bApplyConfig    : BOOL;             (* Rising edge: reconnect with new config *)

    (* ── Manual publish command ───────────────────────── *)
    bPublish        : BOOL;             (* Rising edge: publish sPubPayload       *)
    sPubTopic       : STRING(255);      (* Manual publish topic                   *)
    sPubPayload     : STRING(2048);     (* Manual publish payload                 *)

    (* ── Subscribe command ────────────────────────────── *)
    bSubscribe      : BOOL;             (* Rising edge: subscribe to sSubTopic    *)
    sSubTopic       : STRING(255) := stConfig.SubscribeTopic;      (* Topic to subscribe                     *)
	sPayloadRcv     : STRING(255);     (* Manual publish payload                 *)
	sTopicRcv      	: STRING(255);
	

    (* ── Unsubscribe command ──────────────────────────── *)
    bUnsubscribe    : BOOL;             (* Rising edge: unsubscribe topic         *)
    sUnsubTopic     : STRING(255);      (* Topic to unsubscribe                   *)

    (* ── Cyclic status publishing ─────────────────────── *)
    bEnableStatusPublish : BOOL;        (* TRUE = publish status JSON cyclically  *)
    tStatusPublishTime   : TIME;        (* Example: T#10S                         *)
    sStatusTopic         : STRING(255); (* Example: 'irrigation/status'           *)

    (* ── System data for outgoing JSON ────────────────── *)
    rValveSetpoint       : ARRAY[1..3] OF REAL;
    rValveActual         : ARRAY[1..3] OF REAL;
    sValveSource         : ARRAY[1..3] OF STRING(32);
    rTemperature_C       : REAL;
    rWaterLevel_Percent  : REAL;
    sTimestamp           : STRING(64);
END_VAR


VAR_OUTPUT
    (* ── Connection status ────────────────────────────── *)
    bConnected      : BOOL;             (* TRUE when broker is connected          *)
    bError          : BOOL;             (* TRUE on MQTT error / reconnect state   *)
    nErrorCode      : HRESULT;          (* MQTT HRESULT error code                *)
    sErrorMsg       : STRING(128);      (* Human readable error message           *)

    (* ── Subscribed topic list for HMI ────────────────── *)
    aSubscribedTopic :  STRING(255); //ARRAY[1..20] OF STRING(255);
    nSubscribedCount  : UINT;

    (* ── Command feedback flags ───────────────────────── *)
    bPublishDone      : BOOL;           (* TRUE for one cycle after publish call  *)
    bSubscribeDone    : BOOL;           (* TRUE for one cycle after subscribe     *)
    bUnsubscribeDone  : BOOL;           (* TRUE for one cycle after unsubscribe   *)

    (* ── Incoming command outputs ─────────────────────── *)
    bNewRemoteCommand : BOOL;           (* TRUE for one cycle after valid JSON    *)
    rMqttValveSetpoint : ARRAY[1..3] OF REAL;

    sLastRxTopic      : STRING(255);    (* Last received topic                    *)
    sLastRxPayload    : STRING(2048);   (* Last received payload                  *)

    (* ── Outgoing JSON preview for HMI/debug ──────────── *)
    sJsonStatusPayload : STRING(2048);
END_VAR


VAR
    (* ── MQTT client ──────────────────────────────────── *)
    fbMqttClient : FB_IotMqttClient;
	fbMessageQueue : FB_IotMqttMessageQueue;
	fbMessage      : FB_IotMqttMessage;

    (* ── Connection state machine ─────────────────────── *)
    eState : E_MqttManagerState := E_MqttManagerState.DISABLED;

    (* ── Edge detection ───────────────────────────────── *)
    rtApplyConfig : R_TRIG;
    rtPublish     : R_TRIG;
    rtSubscribe   : R_TRIG;
    rtUnsubscribe : R_TRIG;

    (* ── Timers ───────────────────────────────────────── *)
    tonReconnect     : TON;
    tonStatusPublish : TON;

    (* ── Internal flags ───────────────────────────────── *)
    bConnectCmd : BOOL;
    bReconnectAfterDisconnect : BOOL;

    i : UINT;
    bTopicFound : BOOL;
	
	
    fbJson           : FB_JsonDomParser;
    fbJsonDataType   : FB_JsonReadWriteDatatype;

    (* Incoming *)
    stCmdRecv        : ST_MQTT_Command;

    (* Outgoing *)
    //stStatus         : ST_IrrigationStatus;
	
	bSuccess : BOOL;
	
END_VAR

(* ============================================================
   EDGE DETECTION
   ------------------------------------------------------------
   Convert push-button BOOLs into 1-cycle pulses.
   Example: if bPublish stays TRUE for multiple cycles,
   we still trigger exactly one publish action.
   ============================================================ *)

rtApplyConfig(CLK := bApplyConfig);
rtPublish(CLK := bPublish);
rtSubscribe(CLK := bSubscribe);
rtUnsubscribe(CLK := bUnsubscribe);


(* ============================================================
   RESET ONE-CYCLE FEEDBACK FLAGS
   ============================================================ *)

bPublishDone := FALSE;
bSubscribeDone := FALSE;
bUnsubscribeDone := FALSE;
bNewRemoteCommand := FALSE;


(* ============================================================
   DEFAULT MQTT CONNECT COMMAND

   IMPORTANT:
   Do NOT permanently call Execute(TRUE).
   TRUE  = connect / stay connected
   FALSE = disconnect
   ============================================================ *)

bConnectCmd := FALSE;


(* ============================================================
   CONNECTION STATE MACHINE
   ------------------------------------------------------------
   State intent:
   DISABLED       -> MQTT off by operator
   CONNECTING     -> apply config + request connection
   CONNECTED      -> normal operation (rx/tx)
   DISCONNECTING  -> clean stop before disable/reconfigure
   WAIT_RECONNECT -> back-off timer to avoid fast retry loop
   ============================================================ *)

CASE eState OF

    (* --------------------------------------------------------
       DISABLED

       MQTT is disabled.
       Wait until operator/system sets bEnable = TRUE.
       -------------------------------------------------------- *)
    DISABLED:

        sErrorMsg := '';
        bReconnectAfterDisconnect := FALSE;

        IF bEnable THEN
            eState := CONNECTING;
        END_IF


    (* --------------------------------------------------------
       CONNECTING

       Apply MQTT configuration and request connection.
       Configuration must be assigned before Execute(TRUE).
       -------------------------------------------------------- *)
    CONNECTING:

        fbMqttClient.sHostName     := stConfig.sBrokerAddress;
        fbMqttClient.nHostPort     := stConfig.nPort;
        fbMqttClient.sClientId     := stConfig.sClientId;
        fbMqttClient.sUserName     := stConfig.sUsername;
        fbMqttClient.sUserPassword := stConfig.sPassword;
		fbMqttClient.ipMessageQueue := fbMessageQueue;
		

        bConnectCmd := TRUE;

        IF fbMqttClient.bConnected THEN
            sErrorMsg := '';
            eState := CONNECTED;

        ELSIF fbMqttClient.bError THEN
            sErrorMsg := 'MQTT connect failed. Check broker, port, username/password.';
            eState := WAIT_RECONNECT;
        END_IF


    (* --------------------------------------------------------
       CONNECTED

       MQTT connection is active.
       Monitor enable, config changes, and connection loss.
       -------------------------------------------------------- *)
    CONNECTED:

        bConnectCmd := TRUE;

        IF NOT bEnable THEN
            bReconnectAfterDisconnect := FALSE;
            eState := DISCONNECTING;

        ELSIF rtApplyConfig.Q THEN
            (* Config changed, so disconnect first then reconnect. *)
            bReconnectAfterDisconnect := TRUE;
            eState := DISCONNECTING;

        ELSIF NOT fbMqttClient.bConnected THEN
            (* Unexpected connection loss. *)
            sErrorMsg := 'MQTT connection lost. Reconnecting...';
            eState := WAIT_RECONNECT;
        END_IF


    (* --------------------------------------------------------
       DISCONNECTING

       Execute(FALSE) allows client to disconnect.
       After disconnect:
         • reconnect if config was changed
         • otherwise go to disabled
       -------------------------------------------------------- *)
    DISCONNECTING:

        bConnectCmd := FALSE;

        IF NOT fbMqttClient.bConnected THEN

            IF bEnable AND bReconnectAfterDisconnect THEN
                bReconnectAfterDisconnect := FALSE;
                eState := CONNECTING;
            ELSE
                eState := DISABLED;
            END_IF

        END_IF


    (* --------------------------------------------------------
       WAIT_RECONNECT

       Back-off delay before trying connection again.
       -------------------------------------------------------- *)
    WAIT_RECONNECT:

        bConnectCmd := FALSE;

        tonReconnect(IN := TRUE, PT := stConfig.tReconnectDelay);

        IF NOT bEnable THEN
            tonReconnect(IN := FALSE);
            eState := DISABLED;

        ELSIF tonReconnect.Q THEN
            tonReconnect(IN := FALSE);
            eState := CONNECTING;
        END_IF

END_CASE


(* ============================================================
   EXECUTE MQTT CLIENT

   Must be called every PLC cycle.
   If skipped, MQTT communication and queued message handling stop.
   ============================================================ *)

fbMqttClient.Execute(bConnectCmd);

IF fbMessageQueue.nQueuedMessages > 0 THEN 
    IF fbMessageQueue.Dequeue(fbMessage:=fbMessage) THEN
        fbMessage.GetTopic(pTopic:=ADR(sTopicRcv), nTopicSize:=SIZEOF(sTopicRcv) );
		fbMessage.GetPayload(pPayload:=ADR(sPayloadRcv), nPayloadSize:=SIZEOF(sPayloadRcv), bSetNullTermination:=TRUE);
        bSuccess := fbJsonDataType.SetSymbolFromJson(sPayloadRcv, 'ST_MQTT_COMMAND', SIZEOF(stCmdRecv), ADR(stCmdRecv));
		IF bSuccess THEN
            bNewRemoteCommand := TRUE; // Trigger a flag for other parts of your program
			rMqttValveSetpoint[1] := LIMIT(0.0, DINT_TO_REAL(stCmdRecv.Valve1), 100.0);
			rMqttValveSetpoint[2] := LIMIT(0.0, DINT_TO_REAL(stCmdRecv.Valve2), 100.0);
			rMqttValveSetpoint[3] := LIMIT(0.0, DINT_TO_REAL(stCmdRecv.Valve3), 100.0);
			sLastRxTopic := sTopicRcv;
			sLastRxPayload := sPayloadRcv;
        END_IF
		
	END_IF
END_IF
(* ============================================================
   MANUAL PUBLISH

   Sends sPubPayload to sPubTopic on rising edge of bPublish.
   ============================================================ *)

IF fbMqttClient.bConnected AND rtPublish.Q THEN

    (* Build latest status JSON. *)
    BuildStatusJson();

    fbMqttClient.Publish(
        sTopic       :=  stConfig.sMainTopic,   //sPubTopic,
        pPayload     := ADR(sJsonStatusPayload),
        nPayloadSize := LEN(sJsonStatusPayload),
        eQoS         := TcIotMqttQos.AtMostOnceDelivery,
        bRetain      := TRUE
    );

    bPublishDone := TRUE;
END_IF


(* ============================================================
   SUBSCRIBE TO TOPIC

   TF6701 does not automatically give you a topic list.
   Therefore, this FB stores subscribed topics manually.
   ============================================================ *)

IF fbMqttClient.bConnected AND rtSubscribe.Q THEN

    IF NOT bSubscribeDone THEN
		bSubscribeDone := fbMqttClient.Subscribe(sTopic := sSubTopic, eQoS := TcIotMqttQos.AtMostOnceDelivery);
		IF bSubscribeDone THEN
			aSubscribedTopic := sSubTopic;
			nSubscribedCount := 1;
		END_IF
	END_IF
	

   // bTopicFound := FALSE;
	

(*    (* Check if topic already exists in list. *)
    FOR i := 1 TO 20 DO
        IF aSubscribedTopics[i] = sSubTopic THEN
            bTopicFound := TRUE;
        END_IF
    END_FOR

    (* Add topic to first empty slot. *)
    IF NOT bTopicFound THEN
        FOR i := 1 TO 20 DO
            IF aSubscribedTopics[i] = '' THEN
                aSubscribedTopics[i] := sSubTopic;
                nSubscribedCount := nSubscribedCount + 1;
                EXIT;
            END_IF
        END_FOR
    END_IF
*)
    
END_IF


(* ============================================================
   UNSUBSCRIBE FROM TOPIC

   Removes topic from MQTT broker subscription and local list.
   ============================================================ *)

IF fbMqttClient.bConnected AND rtUnsubscribe.Q THEN

    fbMqttClient.Unsubscribe(
        sTopic := sUnsubTopic
    );

        IF aSubscribedTopic = sUnsubTopic THEN
            aSubscribedTopic := '';

        END_IF
    bUnsubscribeDone := TRUE;
END_IF

(* ============================================================
   CYCLIC STATUS JSON PUBLISH

   Timer-driven telemetry publish for dashboards/history.

   Builds JSON similar to your CSV row and publishes it.
   Example topic:
     irrigation/status
   ============================================================ *)

tonStatusPublish(
    IN := bEnableStatusPublish AND fbMqttClient.bConnected,
    PT := tStatusPublishTime
);

IF tonStatusPublish.Q THEN

    (* Reset timer to create repeating pulse. *)
    tonStatusPublish(IN := FALSE);

    (* Build latest status JSON. *)
    BuildStatusJson();

    (* Publish JSON status. *)
    fbMqttClient.Publish(
        sTopic       := sStatusTopic,
        pPayload     := ADR(sJsonStatusPayload),
        nPayloadSize := LEN(sJsonStatusPayload),
        eQoS         := TcIotMqttQos.AtMostOnceDelivery,
        bRetain      := FALSE
    );

END_IF

(* ============================================================
   OUTPUT STATUS
   ============================================================ *)

bConnected := fbMqttClient.bConnected;
nErrorCode := fbMqttClient.hrErrorCode;

bError := fbMqttClient.bError OR (eState = WAIT_RECONNECT);

IF NOT bError THEN
    nErrorCode := 0;
END_IF

(*
============================================================
METHOD: BuildStatusJson
============================================================

PURPOSE
  Builds outgoing JSON payload similar to the CSV row.

OUTPUT
  sJsonStatusPayload

EXAMPLE
  {
    "timestamp":"2026-04-24 12:30:00",
    "valve_1_setpoint":20.0,
    "valve_1_actual":19.8,
    "valve_1_source":"MQTT",
    ...
  }
============================================================
*)

METHOD BuildStatusJson
VAR
    sTemp : STRING(2048);
END_VAR
sTemp := '{';

sTemp := CONCAT(sTemp, '"timestamp":"');
sTemp := CONCAT(sTemp, sTimestamp);
sTemp := CONCAT(sTemp, '"');

sTemp := CONCAT(sTemp, ',"valve_1_setpoint":');
sTemp := CONCAT(sTemp, REAL_TO_STRING(rValveSetpoint[1]));

sTemp := CONCAT(sTemp, ',"valve_1_actual":');
sTemp := CONCAT(sTemp, REAL_TO_STRING(rValveActual[1]));

sTemp := CONCAT(sTemp, ',"valve_1_source":"');
sTemp := CONCAT(sTemp, sValveSource[1]);
sTemp := CONCAT(sTemp, '"');

sTemp := CONCAT(sTemp, ',"valve_2_setpoint":');
sTemp := CONCAT(sTemp, REAL_TO_STRING(rValveSetpoint[2]));

sTemp := CONCAT(sTemp, ',"valve_2_actual":');
sTemp := CONCAT(sTemp, REAL_TO_STRING(rValveActual[2]));

sTemp := CONCAT(sTemp, ',"valve_2_source":"');
sTemp := CONCAT(sTemp, sValveSource[2]);
sTemp := CONCAT(sTemp, '"');

sTemp := CONCAT(sTemp, ',"valve_3_setpoint":');
sTemp := CONCAT(sTemp, REAL_TO_STRING(rValveSetpoint[3]));

sTemp := CONCAT(sTemp, ',"valve_3_actual":');
sTemp := CONCAT(sTemp, REAL_TO_STRING(rValveActual[3]));

sTemp := CONCAT(sTemp, ',"valve_3_source":"');
sTemp := CONCAT(sTemp, sValveSource[3]);
sTemp := CONCAT(sTemp, '"');

sTemp := CONCAT(sTemp, ',"temperature_c":');
sTemp := CONCAT(sTemp, REAL_TO_STRING(rTemperature_C));

sTemp := CONCAT(sTemp, ',"water_level_percent":');
sTemp := CONCAT(sTemp, REAL_TO_STRING(rWaterLevel_Percent));

sTemp := CONCAT(sTemp, '}');

sJsonStatusPayload := sTemp;
END_METHOD

(*
============================================================
METHOD: GetClientRef
============================================================

PURPOSE
  Returns reference to internal MQTT client.

USE
  Other FBs can use this reference for advanced MQTT handling.
============================================================
*)

METHOD GetClientRef : REFERENCE TO FB_IotMqttClient


GetClientRef REF= fbMqttClient;
END_METHOD

END_FUNCTION_BLOCK
